// TIA Portal V16 export
// export: Created 2021-11-12T13:31:13.744891Z, ExportSetting WithDefaults, DisplayName Totally Integrated Automation Portal, DisplayVersion V16 Update 3, DisplayName TIA Portal Version Control Interface, DisplayVersion V16 Update 2, DisplayName TIA Portal Openness, DisplayVersion V16 Update 3, DisplayName SINAMICS Startdrive Advanced, DisplayVersion V16 Update 5, DisplayName SINAMICS Startdrive G130, G150, S120, S150, SINAMICS MV, S210, DisplayVersion V16 Update 5, DisplayName SINAMICS Startdrive G110M, G120, G120C, G120D, G120P, G115D, DisplayVersion V16 Update 5, DisplayName STEP 7 Professional, DisplayVersion V16 Update 3, DisplayName STEP 7 Safety, DisplayVersion V16, DisplayName WinCC UA Professional, DisplayVersion V16 Update 3
FUNCTION_BLOCK "STD_OnOff"   // FB60, LAD
{ S7_Optimized_Access := 'TRUE' }
VERSION : 0.1
// stored: AutoNumber true, IsIECCheckEnabled false, IsRetainMemResEnabled false, MemoryReserve 100, SetENOAutomatically false, UDAEnableTagReadback false
   VAR_INPUT
      IB_OnOff_1 : Bool;   // Tlačítko zap / vyp - první
      IB_OnOff_2 : Bool;   // Tlačítko zap / vyp - druhé
      IB_OnOff_3 : Bool;   // Tlačítko zap / vyp - třetí
   END_VAR
   VAR_OUTPUT
      OB_On : Bool;   // Akční člen
   END_VAR
   VAR
      SB_Help : Bool;   // Pomocná paměť
   END_VAR
BEGIN

REGION Network 1: On / Off
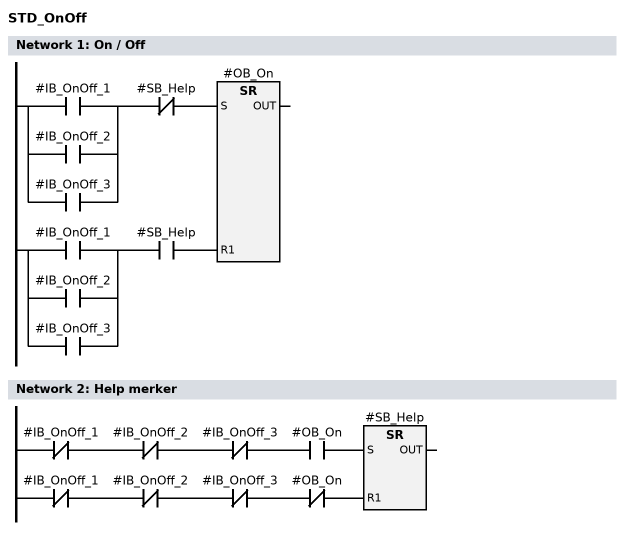
   RUNG wire#powerrail
      Contact( #IB_OnOff_1 )
      wire#w1
      I_Contact( #SB_Help )
      S_SR(operand := #OB_On, r1 := wire#w3)
   END_RUNG
   RUNG wire#powerrail
      Contact( #IB_OnOff_2 )
   END_RUNG wire#w1
   RUNG wire#powerrail
      Contact( #IB_OnOff_3 )
   END_RUNG wire#w1
   RUNG wire#powerrail
      Contact( #IB_OnOff_1 )
      wire#w2
      Contact( #SB_Help )
   END_RUNG wire#w3
   RUNG wire#powerrail
      Contact( #IB_OnOff_2 )
   END_RUNG wire#w2
   RUNG wire#powerrail
      Contact( #IB_OnOff_3 )
   END_RUNG wire#w2
   // the same network as SCL:
   IF (#IB_OnOff_1 OR #IB_OnOff_2 OR #IB_OnOff_3) AND NOT #SB_Help THEN
       #OB_On := TRUE;   // SR flip-flop
   END_IF;
   IF (#IB_OnOff_1 OR #IB_OnOff_2 OR #IB_OnOff_3) AND #SB_Help THEN #OB_On := FALSE; END_IF;
END_REGION

REGION Network 2: Help merker
   RUNG wire#powerrail
      I_Contact( #IB_OnOff_1 )
      I_Contact( #IB_OnOff_2 )
      I_Contact( #IB_OnOff_3 )
      Contact( #OB_On )
      S_SR(operand := #SB_Help, r1 := wire#w1)
   END_RUNG
   RUNG wire#powerrail
      I_Contact( #IB_OnOff_1 )
      I_Contact( #IB_OnOff_2 )
      I_Contact( #IB_OnOff_3 )
      I_Contact( #OB_On )
   END_RUNG wire#w1
   // the same network as SCL:
   IF NOT #IB_OnOff_1 AND NOT #IB_OnOff_2 AND NOT #IB_OnOff_3 AND #OB_On THEN
       #SB_Help := TRUE;   // SR flip-flop
   END_IF;
   IF NOT #IB_OnOff_1 AND NOT #IB_OnOff_2 AND NOT #IB_OnOff_3 AND NOT #OB_On THEN #SB_Help := FALSE; END_IF;
END_REGION
END_FUNCTION_BLOCK
